(* IEC 61131-3 sources: Codesys/ddyut/src (part 2) *)

(* ---- FB_FountainSchedule.st ---- *)
(* ================================================================
   FB_FountainSchedule — Расписание Фонтана (свет + насосы)
   === ДДЮТ:ИЗМЕНЕНО (round 2) === У СВЕТА и НАСОСОВ теперь РАЗНОЕ
   число режимов и РАЗНАЯ кодировка — не путать порядок!

   СВЕТ (Light_Mode, UDINT, 4 положения):
     0 = АВТО   — включение по фиксированному расписанию
                  (Light_On_Hour/Minute_Weekday/Weekend), выключение
                  — общий Off_Hour/Minute (будни/выходные)
     1 = ВКЛ    — горит постоянно, не выключается никогда
     2 = ВЫКЛ   — не включается никогда
     3 = АСТРО  — включение по расчёту заката (Sunset_Hour/Minute
                  от FB_SunsetRelay), выключение — тот же общий
                  Off_Hour/Minute

   НАСОСЫ (Pump_Mode, UDINT, 3 положения — БЕЗ режима "Астро"):
     0 = АВТО   — включение по фиксированному расписанию
                  (Pump_On_Hour/Minute_Weekday/Weekend), выключение
                  — тот же общий Off_Hour/Minute
     1 = ВКЛ    — работает постоянно, не выключается никогда
     2 = ВЫКЛ   — не включается никогда

   === ДДЮТ:ИЗМЕНЕНО === Раньше (round 1) у обоих было по 4
   одинаковых положения (0=Астро,1=Авто,2=Вкл,3=Выкл), полная
   симметрия. По итогам практики решили, что насосам "Астро" не
   нужен — оставили только 3 положения, и заодно поменяли порядок
   у света (Авто теперь 0, Астро — последний, 3). Если переносишь
   в другой проект — ПЕРЕПРОВЕРЬ кодировку, она несимметричная.

   ВАЖНО: это ВНУТРЕННИЙ выбор — работает только когда ВНЕШНИЙ
   селектор узла (GVL_Fountain.iLightSelect / iPumpSelect, экран
   "Свет/Насосы") стоит в положении "Авто" (=2). При "Ручной пуск"
   (=0) и "Выкл" (=1) на внешнем селекторе — этот блок и его режимы
   вообще не участвуют в управлении DO1/DO9.

   ================================================================
   ФЛАГИ ВИДИМОСТИ ДЛЯ ЭКРАНА — единая схема имён:
   Объект_ЧтоПоказывает (Light_/Pump_ + ShowInputFields/
   ShowComputedTime/ShowAlwaysOnText/ShowAlwaysOffText)

   СВЕТ (4 положения, 0=Авто,1=Вкл,2=Выкл,3=Астро):
   Light_ShowInputFields  = TRUE при Режим=0 (Авто) — поля ручного
     ввода расписания (Light_On_Hour/Minute_Weekday/Weekend).
   Light_ShowComputedTime = TRUE при Режим=0 (Авто) ИЛИ Режим=3
     (Астро) — число результата (Light_On_Result_Hour/Minute).
   Light_ShowAlwaysOnText  = TRUE при Режим=1 (Вкл) — текст
     "Свет Вкл ручн".
   Light_ShowAlwaysOffText = TRUE при Режим=2 (Выкл) — текст
     "Свет Выкл ручн".

   НАСОСЫ (3 положения, 0=Авто,1=Вкл,2=Выкл — своя кодировка!):
   Pump_ShowInputFields  = TRUE при Режим=0 (Авто) — поля ручного
     ввода расписания (Pump_On_Hour/Minute_Weekday/Weekend).
   Pump_ShowComputedTime = TRUE при Режим=0 (Авто) — число
     результата. У насосов больше НЕТ режима "Астро" — этот флаг
     истинен только в одном положении, не в двух, как у света.
   Pump_ShowAlwaysOnText  = TRUE при Режим=1 (Вкл) — текст
     "Насосы Вкл ручн".
   Pump_ShowAlwaysOffText = TRUE при Режим=2 (Выкл) — текст
     "Насосы Выкл ручн".

   ---- ОБЩИЕ ПОЛЯ ВЫКЛЮЧЕНИЯ (Off_Result_Hour/Minute — результат,
   и Off_Hour/Minute_Weekday/Weekend — поля ручного ввода уставок) ----
   Актуальны (должны быть видны), если ХОТЯ БЫ ОДИН из двух объектов
   (свет ИЛИ насос) сейчас работает по времени — то есть находится
   в режиме, где Xxx_ShowComputedTime истинен. Если оба постоянно
   "Вкл"/"Выкл" — время выключения нигде не используется, поля
   можно скрыть.

   Off_Time_Visible = Light_ShowComputedTime ИЛИ Pump_ShowComputedTime

   Привязать «Видимость» ко ВСЕМ 6 полям сразу (один и тот же провод
   на несколько свойств «Видимость» — это нормально):
     Off_Result_Hour, Off_Result_Minute,
     Off_Hour_Weekday, Off_Minute_Weekday,
     Off_Hour_Weekend, Off_Minute_Weekend
   ================================================================ *)

FUNCTION_BLOCK FB_FountainSchedule

VAR_INPUT
    (* --- От FB_SunsetRelay --- *)
    Sunset_Auto         : BOOL;
    Sunset_Hour         : UDINT;
    Sunset_Minute       : UDINT;
    IsWeekend           : BOOL;

    (* --- Селектор режима СВЕТА: 0=Авто,1=Вкл,2=Выкл,3=Астро --- *)
    Light_Mode          : UDINT;

    (* --- Ручное расписание СВЕТА (режим 0=Авто): включение --- *)
    Light_On_Hour_Weekday   : UDINT;
    Light_On_Minute_Weekday : UDINT;
    Light_On_Hour_Weekend   : UDINT;
    Light_On_Minute_Weekend : UDINT;

    (* --- Выключение (общее для света и насосов) --- *)
    Off_Hour_Weekday    : UDINT;
    Off_Minute_Weekday  : UDINT;
    Off_Hour_Weekend    : UDINT;
    Off_Minute_Weekend  : UDINT;

    (* --- Селектор режима НАСОСОВ: 0=Авто,1=Вкл,2=Выкл (БЕЗ Астро) --- *)
    Pump_Mode                : UDINT;

    (* --- Ручное расписание НАСОСОВ (режим 0=Авто): включение --- *)
    Pump_On_Hour_Weekday    : UDINT;
    Pump_On_Minute_Weekday  : UDINT;
    Pump_On_Hour_Weekend    : UDINT;
    Pump_On_Minute_Weekend  : UDINT;

    (* --- Текущее время --- *)
    Sys_Hour            : UDINT;
    Sys_Minute          : UDINT;
END_VAR

VAR_OUTPUT
    Light_Out             : BOOL;   (* ВЫХОД на освещение (DO)                *)
    Pump_Out               : BOOL;   (* ВЫХОД на насосы фонтана (DO)           *)

    (* Итоговое время включения СВЕТА на сегодня — для экрана.
       В режимах 1/2 (Вкл/Выкл) содержит 0:00 (заглушка) — привязать
       видимость к Light_ShowComputedTime, чтобы не показывать её.  *)
    Light_On_Result_Hour   : UDINT;
    Light_On_Result_Minute : UDINT;

    (* Итоговое время включения НАСОСОВ на сегодня — для экрана.
       Аналогично, заглушка 0:00 в режимах 1/2 (Вкл/Выкл).          *)
    Pump_On_Result_Hour     : UDINT;
    Pump_On_Result_Minute   : UDINT;

    (* Единое время ВЫКЛЮЧЕНИЯ — общее поле для света и насосов *)
    Off_Result_Hour         : UDINT;
    Off_Result_Minute       : UDINT;

    (* --- Флаги видимости: СВЕТ (0=Авто,1=Вкл,2=Выкл,3=Астро) --- *)
    Light_ShowInputFields    : BOOL;  (* Режим=0(Авто) → поля ручного ввода *)
    Light_ShowComputedTime   : BOOL;  (* Режим=0(Авто) или 3(Астро) → число результата *)
    Light_ShowAlwaysOnText   : BOOL;  (* Режим=1(Вкл) → текст "Свет Вкл ручн" *)
    Light_ShowAlwaysOffText  : BOOL;  (* Режим=2(Выкл) → текст "Свет Выкл ручн" *)

    (* --- Флаги видимости: НАСОСЫ (0=Авто,1=Вкл,2=Выкл, своя кодировка) --- *)
    Pump_ShowInputFields     : BOOL;  (* Режим=0(Авто) → поля ручного ввода *)
    Pump_ShowComputedTime    : BOOL;  (* Режим=0(Авто) → число результата (Астро нет) *)
    Pump_ShowAlwaysOnText    : BOOL;  (* Режим=1(Вкл) → текст "Насосы Вкл ручн" *)
    Pump_ShowAlwaysOffText   : BOOL;  (* Режим=2(Выкл) → текст "Насосы Выкл ручн" *)

    (* Комбинированный флаг для полей времени ВЫКЛЮЧЕНИЯ фонтана
       (Off_Result_Hour/Minute И Off_Hour/Minute_Weekday/Weekend).
       TRUE если хотя бы один из объектов (свет ИЛИ насос) сейчас
       работает по времени.                                        *)
    Off_Time_Visible          : BOOL;
END_VAR

VAR
    now_total_min       : UDINT;
    light_on_min         : UDINT;
    light_off_min        : UDINT;
    pump_on_min           : UDINT;
    pump_off_min          : UDINT;
    off_today_min         : UDINT;  (* Общее время выключения на сегодня (мин) *)
END_VAR

(* ----------------------------------------------------------------
   Текущее время в минутах от 0:00
   ---------------------------------------------------------------- *)
now_total_min := Sys_Hour * 60 + Sys_Minute;

(* Общее время выключения на сегодня (будни/выходные) — используется
   и светом, и насосами, в любом режиме, где это осмысленно          *)
IF IsWeekend THEN
    off_today_min := Off_Hour_Weekend * 60 + Off_Minute_Weekend;
ELSE
    off_today_min := Off_Hour_Weekday * 60 + Off_Minute_Weekday;
END_IF;

(* ================================================================
   СВЕТ — 4 положения: 0=Авто,1=Вкл,2=Выкл,3=Астро
   ================================================================ *)

(* --- Light_Out по режиму --- *)
IF Light_Mode = 0 THEN
    (* АВТО: фиксированное расписание будни/выходные *)
    IF IsWeekend THEN
        light_on_min := Light_On_Hour_Weekend * 60 + Light_On_Minute_Weekend;
    ELSE
        light_on_min := Light_On_Hour_Weekday * 60 + Light_On_Minute_Weekday;
    END_IF;
    light_off_min := off_today_min;

    IF light_off_min > light_on_min THEN
        Light_Out := (now_total_min >= light_on_min) AND (now_total_min < light_off_min);
    ELSE
        Light_Out := (now_total_min >= light_on_min) OR (now_total_min < light_off_min);
    END_IF;

ELSIF Light_Mode = 1 THEN
    Light_Out := TRUE;   (* ВКЛ: горит постоянно *)

ELSIF Light_Mode = 3 THEN
    (* АСТРО: закат → общий Off *)
    light_on_min  := Sunset_Hour * 60 + Sunset_Minute;
    light_off_min := off_today_min;

    IF light_off_min > light_on_min THEN
        Light_Out := (now_total_min >= light_on_min) AND (now_total_min < light_off_min);
    ELSE
        Light_Out := (now_total_min >= light_on_min) OR (now_total_min < light_off_min);
    END_IF;

ELSE
    Light_Out := FALSE;  (* ВЫКЛ (2) или некорректное значение *)
END_IF;

(* --- Light_On_Result --- *)
IF Light_Mode = 0 THEN
    IF IsWeekend THEN
        Light_On_Result_Hour   := Light_On_Hour_Weekend;
        Light_On_Result_Minute := Light_On_Minute_Weekend;
    ELSE
        Light_On_Result_Hour   := Light_On_Hour_Weekday;
        Light_On_Result_Minute := Light_On_Minute_Weekday;
    END_IF;
ELSIF Light_Mode = 3 THEN
    Light_On_Result_Hour   := Sunset_Hour;
    Light_On_Result_Minute := Sunset_Minute;
ELSE
    Light_On_Result_Hour   := 0;   (* заглушка, режимы 1/2 (Вкл/Выкл) *)
    Light_On_Result_Minute := 0;
END_IF;

(* --- Флаги видимости СВЕТА --- *)
Light_ShowInputFields   := (Light_Mode = 0);
Light_ShowComputedTime  := (Light_Mode = 0) OR (Light_Mode = 3);
Light_ShowAlwaysOnText  := (Light_Mode = 1);
Light_ShowAlwaysOffText := (Light_Mode = 2);

(* ================================================================
   НАСОСЫ — 3 положения: 0=Авто,1=Вкл,2=Выкл (БЕЗ режима "Астро")
   ================================================================ *)

(* --- Pump_Out по режиму --- *)
IF Pump_Mode = 0 THEN
    (* АВТО: фиксированное расписание будни/выходные *)
    IF IsWeekend THEN
        pump_on_min := Pump_On_Hour_Weekend * 60 + Pump_On_Minute_Weekend;
    ELSE
        pump_on_min := Pump_On_Hour_Weekday * 60 + Pump_On_Minute_Weekday;
    END_IF;
    pump_off_min := off_today_min;

    IF pump_off_min > pump_on_min THEN
        Pump_Out := (now_total_min >= pump_on_min) AND (now_total_min < pump_off_min);
    ELSE
        Pump_Out := (now_total_min >= pump_on_min) OR (now_total_min < pump_off_min);
    END_IF;

ELSIF Pump_Mode = 1 THEN
    Pump_Out := TRUE;   (* ВКЛ: работает постоянно *)

ELSE
    Pump_Out := FALSE;  (* ВЫКЛ (2) или некорректное значение *)
END_IF;

(* --- Pump_On_Result --- *)
IF Pump_Mode = 0 THEN
    IF IsWeekend THEN
        Pump_On_Result_Hour   := Pump_On_Hour_Weekend;
        Pump_On_Result_Minute := Pump_On_Minute_Weekend;
    ELSE
        Pump_On_Result_Hour   := Pump_On_Hour_Weekday;
        Pump_On_Result_Minute := Pump_On_Minute_Weekday;
    END_IF;
ELSE
    Pump_On_Result_Hour   := 0;   (* заглушка, режимы 1/2 (Вкл/Выкл) *)
    Pump_On_Result_Minute := 0;
END_IF;

(* --- Флаги видимости НАСОСОВ --- *)
Pump_ShowInputFields   := (Pump_Mode = 0);
Pump_ShowComputedTime  := (Pump_Mode = 0);
Pump_ShowAlwaysOnText  := (Pump_Mode = 1);
Pump_ShowAlwaysOffText := (Pump_Mode = 2);

(* ================================================================
   ОБЩЕЕ ПОЛЕ Off_Result (время выключения, одно на экране)
   ================================================================ *)
Off_Result_Hour   := off_today_min / 60;
Off_Result_Minute := off_today_min MOD 60;

Off_Time_Visible := Light_ShowComputedTime OR Pump_ShowComputedTime;

(* ---- FB_Pump.st ---- *)
(* ============================================================ *)
(* FB_Pump — управление одним ПЧ ELHART (PUMP/MINI) по Modbus  *)
(* Проект ДДЮТ (на основе Fontan_V1 / Саки Пруд).               *)
(* === ДДЮТ:ИЗМЕНЕНО === Температура (блок 6) — без деления на  *)
(* 10 (регистр 0x0006 на ДДЮТ отдаёт целые °C). См. комментарий  *)
(* в блоке 6 ниже.                                               *)
(* ============================================================ *)

FUNCTION_BLOCK FB_Pump
VAR_INPUT
    eType      : E_PumpType;
    xDebugMode : BOOL;
    xCommError : BOOL;
    xCommUnstable : BOOL;

    xRunCmd      : BOOL;
    rFreqSetHz   : REAL;

    wStatus          : WORD;
    wFaultReg        : WORD;
    wFreqSetRead     : WORD;
    wFreqActual      : WORD;
    wCurrentActual   : WORD;
    wSpeedActual     : WORD;
    wDcVoltage       : WORD;
    wTemperature     : WORD;
    wVoltageActual   : WORD;
    wRuntimeHoursRaw : WORD;
    wAccTimeRawRead        : WORD;
    wDecTimeRawRead        : WORD;
    wMaxFreqRead           : WORD;
    wMinFreqRead           : WORD;
    wMotorRatedCurrentRead : WORD;
    wMotorRatedVoltageRead : WORD;
    wOverCurrentLevelRead  : WORD;
    wOverheatLevelRead     : WORD;
    wOverCurAccRead        : WORD;
    wOverCurrentTimeRead   : WORD;
    wOverVoltProtectRead   : WORD;

    rAccTime_Set            : REAL;
    rDecTime_Set            : REAL;
    rMaxFreq_Set            : REAL;
    rMinFreq_Set            : REAL;
    rMotorRatedCurrent_Set  : REAL;
    rMotorRatedVoltage_Set  : REAL;
    rOverCurrentLevel_A_Set : REAL;
    rOverCurrentTime_Set    : REAL;
    xOverVoltProtect_Set    : BOOL;
    iOverheatLevel_Set      : INT;
    iOverCurAcc_Set         : INT;
END_VAR
VAR_OUTPUT
    wCmd  : WORD;
    wFreq : WORD;
    wAccTimeRawWrite        : WORD;
    wDecTimeRawWrite        : WORD;
    wMaxFreqWrite           : WORD;
    wMinFreqWrite           : WORD;
    wMotorRatedCurrentWrite : WORD;
    wMotorRatedVoltageWrite : WORD;
    wOverCurrentLevelWrite  : WORD;
    wOverCurrentTimeWrite   : WORD;
    wOverVoltProtectWrite   : WORD;
    wOverheatLevelWrite     : WORD;
    wOverCurAccWrite        : WORD;

    xRun       : BOOL;
    xStop      : BOOL;
    xAlarm     : BOOL;
    sState     : WSTRING(50);
    sFaultText : WSTRING(100);
    sTypeText  : WSTRING(20);
    xReverse   : BOOL;

    rFreqSetActHz : REAL;
    rFreqActHz    : REAL;
    rCurrentActA  : REAL;
    rSpeedActRpm  : REAL;
    rDcVoltageV   : REAL;
    iTemperatureC : INT;
    rVoltageActV  : REAL;
    rRuntimeHours : REAL;
    rAccTime_Disp            : REAL;
    rDecTime_Disp            : REAL;
    rMaxFreq_Disp            : REAL;
    rMinFreq_Disp            : REAL;
    rMotorRatedCurrent_Disp  : REAL;
    rMotorRatedVoltage_Disp  : REAL;
    rOverCurrentLevel_A_Disp : REAL;
    iOverCurrentLevel_pct_Disp : INT;
    iOverheatLevel_Disp      : INT;
    iOverCurAcc_Disp         : INT;
    rOverCurrentTime_Disp    : REAL;
    xOverVoltProtect_Disp    : BOOL;
END_VAR
VAR
    rK_Freq         : REAL;
    rFreqLim        : REAL;
    xFaultActive    : BOOL;
    wCleanFaultCode : WORD;
    iFaultCode      : INT;
    rTmp : REAL;
    iTmp : INT;
END_VAR

(* ========================================================= *)
(* 1. Коэффициент пересчёта частоты                          *)
(* PUMP: 0,01 Гц → k=100 | MINI: 0,1 Гц → k=10               *)
(* ========================================================= *)
IF eType = E_PumpType.PUMP THEN
    rK_Freq   := 100.0;
    sTypeText := "EMD-PUMP";
ELSE
    rK_Freq   := 10.0;
    sTypeText := "EMD-MINI v2.1";
END_IF;

(* ========================================================= *)
(* 2. Команда управления и задание частоты (0x2000 / 0x2001) *)
(* ========================================================= *)
rFreqLim := rFreqSetHz;
IF rFreqLim < cMinFreq THEN rFreqLim := cMinFreq; END_IF;
IF rFreqLim > cMaxFreq THEN rFreqLim := cMaxFreq; END_IF;

IF xRunCmd THEN
    wCmd  := 16#000A;
    wFreq := REAL_TO_WORD(rFreqLim * rK_Freq);
ELSE
    wCmd  := 16#0009;
    wFreq := REAL_TO_WORD(rFreqLim * rK_Freq);
END_IF;

(* ========================================================= *)
(* 3. Нет связи → показать и выйти                           *)
(* ========================================================= *)
xStop := FALSE; xRun := FALSE; xAlarm := FALSE;
xReverse := FALSE; xFaultActive := FALSE;

IF xCommError OR xCommUnstable THEN
    xAlarm     := FALSE;
    xStop      := FALSE;
    xRun       := FALSE;
    sState     := "Нет связи с ПЧ";
    sFaultText := "Проверьте RS-485 / адрес / питание ПЧ";
    RETURN;
END_IF;

(* ========================================================= *)
(* 4. Состояние ПЧ по 0x001C                                *)
(* ========================================================= *)
CASE eType OF
    E_PumpType.PUMP:
        xReverse := (wStatus AND 16#0004) <> 0;
        IF (wStatus AND 16#0008) <> 0 THEN
            xAlarm := TRUE; xFaultActive := TRUE; sState := "Авария";
        ELSIF (wStatus AND 16#0001) <> 0 THEN
            xRun := TRUE;
            IF xReverse THEN sState := "Работа (реверс)"; ELSE sState := "Работа"; END_IF;
        ELSE
            xStop := TRUE; sState := "Стоп";
        END_IF;
    E_PumpType.MINI:
        xReverse := (wStatus AND 16#0001) <> 0;
        IF (wStatus AND 16#0002) <> 0 THEN
            xRun := TRUE;
            IF xReverse THEN sState := "Работа (реверс)"; ELSE sState := "Работа"; END_IF;
        ELSE
            xStop := TRUE; sState := "Стоп";
        END_IF;
END_CASE;

(* ========================================================= *)
(* 5. Разбор аварий                                         *)
(* ========================================================= *)
CASE eType OF
    E_PumpType.PUMP:
        IF (wFaultReg AND 16#8000) <> 0 THEN
            xAlarm := TRUE; xRun := FALSE; xStop := FALSE; sState := "Авария";
            wCleanFaultCode := wFaultReg AND 16#7FFF;
            sFaultText := F_FaultCodeToText(eType, wCleanFaultCode);
        ELSE
            sFaultText := "Нет ошибок";
        END_IF;
    E_PumpType.MINI:
        iFaultCode := WORD_TO_INT(wFaultReg);
        IF (iFaultCode > 63) AND ((iFaultCode < 88) OR (iFaultCode > 91)) THEN
            xAlarm := TRUE; xRun := FALSE; xStop := FALSE; sState := "Авария";
            sFaultText := F_FaultCodeToText(eType, wFaultReg);
        ELSE
            sFaultText := "Нет ошибок";
        END_IF;
END_CASE;

(* ========================================================= *)
(* 6. ЧТЕНИЕ реальных значений из ПЧ → _Disp (для показа)    *)
(* ========================================================= *)
rFreqSetActHz := WORD_TO_REAL(wFreqSetRead) / rK_Freq;
rFreqActHz    := WORD_TO_REAL(wFreqActual)  / rK_Freq;
rCurrentActA  := WORD_TO_REAL(wCurrentActual) / 10.0;
rSpeedActRpm  := WORD_TO_REAL(wSpeedActual);
rDcVoltageV   := WORD_TO_REAL(wDcVoltage) / 10.0;

(* === ДДЮТ:ИЗМЕНЕНО === Температура: БЕЗ деления на 10.       *)
(* На Саки регистр 0x0006 отдавал ×10 (0.1°C), на ДДЮТ — уже    *)
(* целые °C (та же марка ПЧ, но другая дискретность регистра —  *)
(* сверено на объекте: /10.0 давало 4°C вместо реальных 40°C).  *)
(* Если на твоём ПЧ регистр всё-таки ×10 — верни /10.0 обратно. *)
iTemperatureC := WORD_TO_INT(wTemperature);

rVoltageActV  := WORD_TO_REAL(wVoltageActual) / 10.0;
rRuntimeHours := WORD_TO_REAL(wRuntimeHoursRaw);

rAccTime_Disp           := WORD_TO_REAL(wAccTimeRawRead) / 10.0;
rDecTime_Disp           := WORD_TO_REAL(wDecTimeRawRead) / 10.0;
rMaxFreq_Disp           := WORD_TO_REAL(wMaxFreqRead) / rK_Freq;
rMinFreq_Disp           := WORD_TO_REAL(wMinFreqRead) / rK_Freq;
rMotorRatedCurrent_Disp := WORD_TO_REAL(wMotorRatedCurrentRead) / 10.0;
rMotorRatedVoltage_Disp := WORD_TO_REAL(wMotorRatedVoltageRead) / 10.0;
iOverCurrentLevel_pct_Disp := WORD_TO_INT(wOverCurrentLevelRead);
IF rMotorRatedCurrent_Disp > 0.0 THEN
    rOverCurrentLevel_A_Disp := (INT_TO_REAL(iOverCurrentLevel_pct_Disp) / 100.0)
                                 * rMotorRatedCurrent_Disp;
ELSE
    rOverCurrentLevel_A_Disp := 0.0;
END_IF;
iOverheatLevel_Disp := WORD_TO_INT(wOverheatLevelRead);
iOverCurAcc_Disp    := WORD_TO_INT(wOverCurAccRead);
rOverCurrentTime_Disp := WORD_TO_REAL(wOverCurrentTimeRead) / 10.0;
xOverVoltProtect_Disp := (wOverVoltProtectRead <> WORD#0);

(* ========================================================= *)
(* 7. ЗАДАНИЕ оператора → регистры ЗАПИСИ (_Set, с валидацией)*)
(* ========================================================= *)
rTmp := rAccTime_Set;
IF rTmp < cMinTime THEN rTmp := cMinTime; ELSIF rTmp > cMaxTime THEN rTmp := cMaxTime; END_IF;
wAccTimeRawWrite := REAL_TO_WORD(rTmp * 10.0);

rTmp := rDecTime_Set;
IF rTmp < cMinTime THEN rTmp := cMinTime; ELSIF rTmp > cMaxTime THEN rTmp := cMaxTime; END_IF;
wDecTimeRawWrite := REAL_TO_WORD(rTmp * 10.0);

rTmp := rMaxFreq_Set;
IF rTmp < 1.0 THEN rTmp := 1.0; ELSIF rTmp > cMaxFreq THEN rTmp := cMaxFreq; END_IF;
wMaxFreqWrite := REAL_TO_WORD(rTmp * rK_Freq);
rTmp := rMinFreq_Set;
IF rTmp < 0.0 THEN rTmp := 0.0; ELSIF rTmp > rMaxFreq_Set THEN rTmp := rMaxFreq_Set; END_IF;
wMinFreqWrite := REAL_TO_WORD(rTmp * rK_Freq);

rTmp := rMotorRatedVoltage_Set;
IF rTmp < 0.0 THEN rTmp := 0.0; ELSIF rTmp > cMaxVoltage THEN rTmp := cMaxVoltage; END_IF;
wMotorRatedVoltageWrite := REAL_TO_WORD(rTmp * 10.0);
rTmp := rMotorRatedCurrent_Set;
IF rTmp < 0.1 THEN rTmp := 0.1; ELSIF rTmp > cMaxCurrent THEN rTmp := cMaxCurrent; END_IF;
wMotorRatedCurrentWrite := REAL_TO_WORD(rTmp * 10.0);

IF rMotorRatedCurrent_Set > 0.0 THEN
    iTmp := REAL_TO_INT((rOverCurrentLevel_A_Set / rMotorRatedCurrent_Set) * 100.0);
ELSE
    iTmp := 0;
END_IF;
IF iTmp < 0 THEN iTmp := 0; ELSIF iTmp > 200 THEN iTmp := 200; END_IF;
wOverCurrentLevelWrite := INT_TO_WORD(iTmp);

rTmp := rOverCurrentTime_Set;
IF rTmp < 0.0 THEN rTmp := 0.0; END_IF;
CASE eType OF
    E_PumpType.PUMP: IF rTmp > 999.9 THEN rTmp := 999.9; END_IF;
    E_PumpType.MINI: IF rTmp > 5.0 THEN rTmp := 5.0; END_IF;
END_CASE;
wOverCurrentTimeWrite := REAL_TO_WORD(rTmp * 10.0);

IF xOverVoltProtect_Set THEN wOverVoltProtectWrite := 1; ELSE wOverVoltProtectWrite := 0; END_IF;

iTmp := iOverheatLevel_Set;
IF iTmp < cMinOverheat THEN iTmp := cMinOverheat; ELSIF iTmp > cMaxOverheat THEN iTmp := cMaxOverheat; END_IF;
wOverheatLevelWrite := INT_TO_WORD(iTmp);

iTmp := iOverCurAcc_Set;
IF iTmp < 0 THEN iTmp := 0; ELSIF iTmp > 200 THEN iTmp := 200; END_IF;
wOverCurAccWrite := INT_TO_WORD(iTmp);

(* ---- FB_SdSpaceGuard.st ---- *)
(* ============================================================ *)
(* FB_SdSpaceGuard — СТОРОЖ МЕСТА НА SD + УДАЛЕНИЕ САМОГО        *)
(*                   СТАРОГО МЕСЯЦА ЖУРНАЛОВ                     *)
(* ============================================================ *)
(* Ёмкость карты приходит на вход udiUsableMB: её определяет сам   *)
(* FB_SdCardSize (читает размер раздела у ядра), а если не вышло — *)
(* берётся номинал из выпадающего списка на экране (iSdCardSize).  *)
(*                                                               *)
(* ЧТО ДЕЛАЕТ ЗА ОДИН ЗАПУСК (фронт xTrigger):                    *)
(*   1. Обходит каталог журналов (DirOpen → DirList → DirClose):  *)
(*      считает, сколько занимают НАШИ журналы и сколько чужие,   *)
(*      и ищет САМЫЙ СТАРЫЙ месяц.                               *)
(*   2. Считает потолок:                                          *)
(*        квота = ёмкость карты − резерв 100 МБ − чужие файлы     *)
(*      То есть журналам достаётся ВСЯ карта, кроме резерва: на   *)
(*      32 ГБ это ~28,9 ГБ, на 2 ГБ ~1,7 ГБ. Ничего не пропадает. *)
(*   3. Если наши журналы переросли квоту — удаляет ТРИ файла     *)
(*      самого старого месяца и повторяет с пункта 1, пока не     *)
(*      уложится.                                                *)
(*                                                               *)
(* ⚠️ В квоту считается объём ТОЛЬКО наших файлов (прошедших       *)
(* разбор F_SdLogMonthKey), а чужие вычитаются из ёмкости — так    *)
(* чей-то архив на карте уменьшает наш потолок, но удалён быть не  *)
(* может. Содержимое ВЛОЖЕННЫХ папок не считается (DirList в       *)
(* глубину не ходит) — папку app.spk1xxm01 с загрузочным           *)
(* приложением (единицы МБ) перекрывает резерв в 100 МБ.           *)
(*                                                               *)
(* ЗАЩИТЫ ОТ УДАЛЕНИЯ ЛИШНЕГО:                                    *)
(*   • Удаляются только имена, ТОЧНО совпавшие с шаблоном         *)
(*     "<префикс>MM-YYYY.log" (разбор в F_SdLogMonthKey).         *)
(*   • Файл текущего месяца (в который идёт запись) не может быть *)
(*     удалён в принципе: кандидат обязан быть СТРОГО СТАРШЕ.     *)
(*   • Сравнение по числовому ключу YYYY*12+MM-1, а не по строке: *)
(*     12-2025 корректно старше 01-2026.                          *)
(*   • Каталоги (deDirEntry.xDirectory) пропускаются целиком.      *)
(*   • Если обход каталога оборвался по лимиту — «самый старый»   *)
(*     недостоверен, и не удаляется НИЧЕГО.                       *)
(*                                                               *)
(* ЕСЛИ УДАЛЯТЬ УЖЕ НЕЧЕГО, А КВОТА ВСЁ РАВНО ПРЕВЫШЕНА           *)
(* (вся история — это один текущий месяц, раздутый дребезгом      *)
(* аварий), поднимается xQuotaStop, и PRG_AlarmLogSD ПРЕКРАЩАЕТ   *)
(* запись на карту. Это последний рубеж: карта не переполнится    *)
(* никогда, фонтан работает, журналы на экране ведутся как        *)
(* обычно. Снимается само при смене месяца, когда раздутый файл   *)
(* станет прошлым и его можно будет удалить. Человек не нужен.    *)
(*                                                               *)
(* ЕДИНИЦЫ. Внутри всё в КиБ (1024 байта), наружу и в пороги — в   *)
(* МиБ (1024 КиБ = 1 048 576 байт). 100 МБ = 104 857 600 байт.    *)
(* Деление целочисленное: оценка свободного всегда чуть ЗАНИЖЕНА, *)
(* то есть чистка срабатывает на доли мегабайта РАНЬШЕ.           *)
(*                                                               *)
(* ФБ асинхронный: один запуск растянут на много циклов ПЛК       *)
(* (каждый ФБ CAA File требует минимум цикл). Пока xBusy = TRUE,  *)
(* PRG_AlarmLogSD не начинает новую запись строки.                *)
(* ============================================================ *)
FUNCTION_BLOCK FB_SdSpaceGuard
VAR_INPUT
    xTrigger      : BOOL;        (* ФРОНТ — выполнить проверку *)
    xForce        : BOOL;        (* уровень, читается при старте: удалить    *)
                                 (* самый старый месяц БЕЗ проверок. Ставится*)
                                 (* автоматически, когда запись на карту не  *)
                                 (* проходит подряд несколько раз (значит,   *)
                                 (* карта реально полна — например, номинал  *)
                                 (* в списке выбран больше настоящего).      *)
    sDir          : STRING(80);  (* каталог журналов, БЕЗ '/' в конце *)
    sPrefix1      : STRING(20);  (* 'alarms-' *)
    sPrefix2      : STRING(20);  (* 'pump_changes-' *)
    sPrefix3      : STRING(20);  (* 'setpoints-' *)
    udiUsableMB   : UDINT;       (* полезная ёмкость карты, МиБ *)
    udiFreeMinMB  : UDINT;       (* резерв свободного места, МиБ (100) *)
    iCurYear      : INT;         (* текущий год  журнала (2000..2199) *)
    iCurMonth     : INT;         (* текущий месяц журнала (1..12) *)
END_VAR
VAR_OUTPUT
    xBusy            : BOOL;
    xDone            : BOOL;      (* импульс 1 цикл по завершении запуска *)
    xQuotaStop       : BOOL;      (* ⛔ писать на SD больше нельзя *)
    udiQuotaMB       : UDINT;     (* сколько реально отдано журналам, МиБ *)
    udiOursMB        : UDINT;     (* занято НАШИМИ журналами, МиБ *)
    udiUsedMB        : UDINT;     (* занято всеми файлами каталога, МиБ *)
    udiForeignMB     : UDINT;     (* занято чужими файлами рядом, МиБ *)
    udiOldestMB      : UDINT;     (* объём самого старого месяца, МиБ *)
    xNothingToDelete : BOOL;      (* чистить надо, а удалять нечего *)
    xFault           : BOOL;      (* карта/каталог недоступны, скан сорван *)
    iDeletedTotal    : INT;       (* удалено файлов с момента старта ПЛК *)
    iDeletedLast     : INT;       (* удалено за последний запуск *)
    sLastDeleted     : STRING(80);(* что удалили последним *)
    iFilesSeen       : INT;       (* файлов в каталоге на последнем скане *)
END_VAR
VAR CONSTANT
    cMaxRounds  : INT := 24;      (* не больше 24 месяцев за один запуск *)
    cMaxEntries : INT := 500;     (* страховка от бесконечного DirList *)
END_VAR
VAR
    iSt        : INT;
    xTrigPrev  : BOOL;
    iRound     : INT;

    fbDirOpen  : FILE.DirOpen;
    fbDirList  : FILE.DirList;
    fbDirClose : FILE.DirClose;
    fbDelete   : FILE.Delete;
    hDir       : FILE.CAA.HANDLE;

    udiUsedKB    : UDINT;   (* все файлы каталога, КиБ (диагностика) *)
    udiOursKB    : UDINT;   (* только наши журналы, КиБ (для квоты) *)
    udiEntryKB   : UDINT;
    udiCurKey    : UDINT;
    udiOldKey    : UDINT;
    udiOldestKB  : UDINT;   (* объём файлов самого старого месяца, КиБ *)
    udiKey       : UDINT;
    xFoundOld    : BOOL;
    xForceRun    : BOOL;
    xOverQuota   : BOOL;
    iEntries     : INT;
    sEntry       : STRING(255);

    iOldYear        : INT;
    iOldMonth       : INT;
    iDelIdx         : INT;
    iDelOkThisRound : INT;
    sDelPath        : STRING(80);
END_VAR

(* ============================================================ *)
(* ЗАПУСК ПО ФРОНТУ                                             *)
(* ============================================================ *)
IF xTrigger AND NOT xTrigPrev AND iSt = 0 THEN
    xForceRun := xForce;      (* режим запуска фиксируем в момент старта *)
    iSt := 10;
END_IF;
xTrigPrev := xTrigger;

xDone := FALSE;
xBusy := (iSt <> 0);

CASE iSt OF

    0:  (* IDLE *)
        ;

    10: (* НАЧАЛО ЗАПУСКА *)
        iRound           := 0;
        iDeletedLast     := 0;
        xNothingToDelete := FALSE;
        xFault           := FALSE;
        iSt := 11;

    11: (* НАЧАЛО РАУНДА — подготовка скана каталога *)
        IF iCurYear < 2000 OR iCurYear > 2199 OR iCurMonth < 1 OR iCurMonth > 12 THEN
            (* без достоверного «сегодня» нельзя понять, какой месяц    *)
            (* трогать нельзя → не удаляем НИЧЕГО                        *)
            xFault := TRUE;
            iSt := 90;
        ELSE
            udiCurKey    := INT_TO_UDINT(iCurYear) * 12 + INT_TO_UDINT(iCurMonth) - 1;
            udiUsedKB    := 0;
            udiOursKB    := 0;
            udiOldKey    := 0;
            udiOldestKB  := 0;
            xFoundOld    := FALSE;
            iEntries     := 0;
            iSt := 12;
        END_IF;

    12: (* DirOpen *)
        fbDirOpen(xExecute := TRUE, sDirName := sDir);
        IF fbDirOpen.xDone THEN
            hDir := fbDirOpen.hDir;
            fbDirOpen(xExecute := FALSE);
            iSt := 13;
        ELSIF fbDirOpen.xError THEN
            fbDirOpen(xExecute := FALSE);
            xFault := TRUE;          (* карты нет / каталог недоступен *)
            iSt := 90;
        END_IF;

    13: (* DirList — по ОДНОЙ записи за вызов, до NO_MORE_ENTRIES *)
        fbDirList(xExecute := TRUE, hDir := hDir);
        IF fbDirList.xDone THEN
            IF NOT fbDirList.deDirEntry.xDirectory THEN
                sEntry := fbDirList.deDirEntry.sEntry;

                (* объём: округляем вверх до КиБ — оценка занятого места     *)
                (* получается чуть больше реальной суммы байт, это в нужную  *)
                (* сторону (реальный расход по кластерам FAT ещё больше)     *)
                udiEntryKB := (fbDirList.deDirEntry.szSize / 1024) + 1;
                udiUsedKB  := udiUsedKB + udiEntryKB;

                (* наш ли это файл и за какой месяц *)
                udiKey := F_SdLogMonthKey(sEntry, sPrefix1);
                IF udiKey = 0 THEN udiKey := F_SdLogMonthKey(sEntry, sPrefix2); END_IF;
                IF udiKey = 0 THEN udiKey := F_SdLogMonthKey(sEntry, sPrefix3); END_IF;

                IF udiKey > 0 THEN
                    (* КВОТА считается только по НАШИМ файлам *)
                    udiOursKB := udiOursKB + udiEntryKB;

                    (* кандидат на удаление — только СТРОГО СТАРШЕ текущего *)
                    IF udiKey < udiCurKey THEN
                        IF NOT xFoundOld OR udiKey < udiOldKey THEN
                            (* нашли месяц старее — объём считаем заново *)
                            udiOldKey   := udiKey;
                            udiOldestKB := udiEntryKB;
                            xFoundOld   := TRUE;
                        ELSIF udiKey = udiOldKey THEN
                            (* ещё один файл того же самого старого месяца *)
                            udiOldestKB := udiOldestKB + udiEntryKB;
                        END_IF;
                    END_IF;
                END_IF;
            END_IF;

            iEntries := iEntries + 1;
            fbDirList(xExecute := FALSE);
            IF iEntries >= cMaxEntries THEN
                (* Каталог не дочитан до конца → «самый старый месяц»         *)
                (* определён по неполному списку и может быть НЕ самым старым. *)
                (* Удалять по недостоверным данным нельзя: закрываем каталог   *)
                (* и выходим с аварией. 500 файлов — это ~13 лет журналов,     *)
                (* столько бывает только если на карте лежит что-то чужое.     *)
                xFault := TRUE;
                iSt := 14;
            END_IF;
        ELSIF fbDirList.xError THEN
            (* штатное окончание обхода = ERROR.NO_MORE_ENTRIES *)
            fbDirList(xExecute := FALSE);
            iSt := 14;
        END_IF;

    14: (* DirClose — закрыть каталог НАДО в любом случае, даже по аварии *)
        fbDirClose(xExecute := TRUE, hDir := hDir);
        IF fbDirClose.xDone OR fbDirClose.xError THEN
            fbDirClose(xExecute := FALSE);
            iFilesSeen := iEntries;
            IF xFault THEN
                iSt := 90;      (* скан недостоверен — ничего не удаляем *)
            ELSE
                iSt := 20;
            END_IF;
        END_IF;

    20: (* ОЦЕНКА: КВОТА *)
        udiUsedMB   := udiUsedKB / 1024;
        udiOursMB   := udiOursKB / 1024;
        udiOldestMB := udiOldestKB / 1024;

        (* --- сколько можно отдать журналам ---                          *)
        (* Вся карта минус резерв минус ЧУЖИЕ файлы, лежащие рядом в том  *)
        (* же каталоге (например, распакованное загрузочное приложение).  *)
        (* ⚠️ Содержимое ВЛОЖЕННЫХ папок не считается — DirList в глубину  *)
        (* не ходит. Папку app.spk1xxm01 с проектом (единицы МБ) с лихвой  *)
        (* перекрывает резерв в 100 МБ.                                   *)
        udiForeignMB := udiUsedMB - udiOursMB;
        IF udiUsableMB > (udiFreeMinMB + udiForeignMB) THEN
            udiQuotaMB := udiUsableMB - udiFreeMinMB - udiForeignMB;
        ELSE
            udiQuotaMB := 0;    (* чужие файлы съели всё — чистимся до дна *)
        END_IF;

        (* --- превышен ли потолок --- *)
        xOverQuota := (udiOursMB > udiQuotaMB);

        iSt := 30;

    30: (* РЕШЕНИЕ: чистить или нет *)
        IF xForceRun OR xOverQuota THEN
            IF xFoundOld THEN
                iOldYear        := UDINT_TO_INT(udiOldKey / 12);
                iOldMonth       := UDINT_TO_INT(udiOldKey MOD 12) + 1;
                iDelIdx         := 1;
                iDelOkThisRound := 0;
                iSt := 40;
            ELSE
                (* Старше текущего месяца ничего нет. Если при этом превышена *)
                (* наша собственная квота — единственный оставшийся способ не *)
                (* переполнить карту — перестать писать. Снимется само на     *)
                (* следующем месяце.                                          *)
                xNothingToDelete := TRUE;
                xQuotaStop       := xOverQuota;
                iSt := 90;
            END_IF;
        ELSE
            (* всё в норме — снимаем запрет записи, если он был *)
            xNothingToDelete := FALSE;
            xQuotaStop       := FALSE;
            iSt := 90;
        END_IF;

    40: (* ИМЯ ОЧЕРЕДНОГО ФАЙЛА САМОГО СТАРОГО МЕСЯЦА *)
        CASE iDelIdx OF
            1: sDelPath := F_SdLogPath(sDir, sPrefix1, iOldYear, iOldMonth);
            2: sDelPath := F_SdLogPath(sDir, sPrefix2, iOldYear, iOldMonth);
            3: sDelPath := F_SdLogPath(sDir, sPrefix3, iOldYear, iOldMonth);
        END_CASE;
        iSt := 41;

    41: (* УДАЛЕНИЕ *)
        fbDelete(xExecute := TRUE, sFileName := sDelPath);
        IF fbDelete.xDone THEN
            fbDelete(xExecute := FALSE);
            iDeletedLast    := iDeletedLast + 1;
            iDeletedTotal   := iDeletedTotal + 1;
            iDelOkThisRound := iDelOkThisRound + 1;
            sLastDeleted    := sDelPath;
            iSt := 42;
        ELSIF fbDelete.xError THEN
            (* файла за этот месяц могло не быть (например, уставки никто    *)
            (* не менял) — это норма, просто идём дальше                     *)
            fbDelete(xExecute := FALSE);
            iSt := 42;
        END_IF;

    42: (* СЛЕДУЮЩИЙ ФАЙЛ ИЛИ СЛЕДУЮЩИЙ РАУНД *)
        IF iDelIdx < 3 THEN
            iDelIdx := iDelIdx + 1;
            iSt := 40;
        ELSE
            iRound    := iRound + 1;
            xForceRun := FALSE;      (* аварийный форс = ровно один месяц *)
            IF iDelOkThisRound = 0 THEN
                (* Скан этот месяц нашёл, а удалить не вышло НИ ОДНОГО файла: *)
                (* карта только для чтения / вынута / имя на ФС отличается     *)
                (* регистром. Повторять раунды бессмысленно — они будут снова  *)
                (* находить тот же месяц. Выходим с аварией, чтобы это увидели.*)
                xFault := TRUE;
                iSt := 90;
            ELSIF iRound >= cMaxRounds THEN
                iSt := 90;
            ELSE
                iSt := 11;           (* пересчитать и, если надо, ещё раз *)
            END_IF;
        END_IF;

    90: (* КОНЕЦ ЗАПУСКА *)
        xDone := TRUE;
        iSt   := 0;

END_CASE;

(* ---- FB_SunsetRelay.st ---- *)
(* ============================================================
   FB_SunsetRelay — Астрономическое реле (расчёт заката)
   === ДДЮТ:ПОРТИРОВАНО (v2, точность до 1 мин) ===
   Единственное техническое отличие от твоего исходника (OwenLogic):
     SYS.COS/SYS.SIN/SYS.TAN/SYS.ACOS → COS/SIN/TAN/ACOS
     (в CODESYS это стандартные функции IEC 61131-3 без префикса
     SYS. — префикс есть только в библиотеке OwenLogic).
   Вся математика, включая поправку на рефракцию (90.833°) и
   алгоритм Зеллера — БЕЗ ИЗМЕНЕНИЙ, как в твоём исходнике.
   Логика:
   - Расчёт времени заката по долготе/широте/часовому поясу
   - Ручная коррекция ±минут (местность: море/горы/рельеф)
   - Выход «Sunset_Auto» = TRUE от заката до времени отключения
   - Точность расчёта: ±1-3 минуты (алгоритм NOAA/Spencer с поправкой
     на атмосферную рефракцию и радиус диска Солнца, угол зенита
     90.833°). Сверено с независимыми источниками для трёх городов
     на 12 месяцев вперёд.
   - Определение будни/выходной (алгоритм Зеллера) — для выбора
     своей пары Off_Hour/Off_Minute, а также выдаётся наружу
     (IsWeekend) для использования в FB_FountainSchedule, чтобы
     не дублировать расчёт дня недели в другом блоке.
   - Доп. выход: сколько осталось до следующей смены состояния

   ВАЖНО: Sunset_Auto — это ТОЛЬКО автоматический расчёт по закату.
   Финальное управление светом (авто/ручной режим) находится в
   отдельном блоке FB_FountainSchedule — туда подаётся Sunset_Auto
   как один из входов.
   ============================================================ *)

FUNCTION_BLOCK FB_SunsetRelay

VAR_INPUT
    (* --- Геокоординаты с экрана --- *)
    Latitude        : REAL;   (* Широта, градусы (пример: 44.59 = Севастополь)  *)
    Longitude       : REAL;   (* Долгота, градусы (пример: 33.52 = Севастополь) *)
    TimeZone        : REAL;   (* Часовой пояс, знаковый! ← выход FB_TimeZoneSelect *)

    (* --- Коррекция заката --- *)
    Sunset_Correct  : UDINT;  (* Ручная коррекция заката, минут (0..60)  *)
    Sunset_Earlier   : BOOL;  (* Направление: TRUE = раньше, FALSE = позже *)

    (* --- Настройки отключения: раздельно будни/выходные --- *)
    Off_Hour_Weekday   : UDINT;  (* Час отключения, будний день      *)
    Off_Minute_Weekday : UDINT;  (* Минута отключения, будний день   *)
    Off_Hour_Weekend   : UDINT;  (* Час отключения, выходной день    *)
    Off_Minute_Weekend : UDINT;  (* Минута отключения, выходной день *)

    (* --- Системное время (привязка к RTC ПР200) --- *)
    Sys_Year        : UDINT;  (* Год (2026)                              *)
    Sys_Month       : UDINT;  (* Месяц (1..12)                           *)
    Sys_Day         : UDINT;  (* День (1..31)                            *)
    Sys_Hour        : UDINT;  (* Часы (0..23)                            *)
    Sys_Minute      : UDINT;  (* Минуты (0..59)                          *)
    Sys_Sec         : UDINT;  (* Секунды (0..59) — для точности          *)
END_VAR

VAR_OUTPUT
    Sunset_Auto     : BOOL;   (* Автоматический расчёт: 1 = должно гореть *)
    Sunset_Hour     : UDINT;  (* Рассчитанный час заката (для экрана)    *)
    Sunset_Minute   : UDINT;  (* Рассчитанная минута заката (для экрана) *)
    DayOfYear       : UDINT;  (* Порядковый день года (диагностика)      *)
    Err_Coord       : BOOL;   (* Ошибка координат (широта за пределами)  *)
    IsWeekend       : BOOL;   (* TRUE = суббота/воскресенье. Выдаётся
                                  наружу для FB_FountainSchedule           *)

    (* --- Сколько осталось до следующего включения --- *)
    Time_Left_H     : UDINT;  (* Осталось ждать: часы                    *)
    Time_Left_M     : UDINT;  (* Осталось ждать: минуты (0–59)           *)
END_VAR

VAR
    (* --- Внутренние переменные расчёта заката --- *)
    i               : UDINT;
    doy             : UDINT;
    lat_rad         : REAL;
    gamma           : REAL;
    eqtime          : REAL;
    decl            : REAL;
    ha              : REAL;
    sunset_utc      : REAL;
    sunset_local    : REAL;
    sunset_total_min : UDINT;
    off_total_min   : UDINT;
    now_total_min   : UDINT;
    diff_min        : UDINT;
    pi              : REAL;
    two_pi          : REAL;
    deg_to_rad      : REAL;
    rad_to_deg      : REAL;
    temp_real       : REAL;
    sunset_corr_real : REAL;
    days_in_month   : ARRAY[1..12] OF UDINT;

    (* --- Внутренние переменные расчёта дня недели (алгоритм Зеллера) --- *)
    zm              : UDINT;  (* Месяц с коррекцией (янв/фев → 13/14 пред. года) *)
    zy              : UDINT;  (* Год с коррекцией                         *)
    zK              : UDINT;  (* Год внутри века (00-99)                  *)
    zJ              : UDINT;  (* Век (число столетий)                     *)
    zh              : UDINT;  (* Результат: 0=Сб,1=Вс,2=Пн,3=Вт,4=Ср,5=Чт,6=Пт *)
END_VAR

(* ============================================================
   ОПРЕДЕЛЕНИЕ ДНЯ НЕДЕЛИ (алгоритм Зеллера, григорианский календарь)
   Выполняется ВСЕГДА, независимо от Err_Coord — не зависит от
   координат, нужно для выбора Off_Hour/Off_Minute и для выдачи
   IsWeekend наружу.
   ============================================================ *)
IF Sys_Month < 3 THEN
    zm := Sys_Month + 12;
    zy := Sys_Year - 1;
ELSE
    zm := Sys_Month;
    zy := Sys_Year;
END_IF;

zK := zy MOD 100;
zJ := zy / 100;

zh := (Sys_Day + (13 * (zm + 1)) / 5 + zK + zK / 4 + zJ / 4 + 5 * zJ) MOD 7;

IsWeekend := (zh = 0) OR (zh = 1);   (* 0=суббота, 1=воскресенье *)

(* Выбор пары Off_Hour/Off_Minute по дню недели *)
IF IsWeekend THEN
    off_total_min := Off_Hour_Weekend * 60 + Off_Minute_Weekend;
ELSE
    off_total_min := Off_Hour_Weekday * 60 + Off_Minute_Weekday;
END_IF;

(* ============================================================
   ТЕЛО БЛОКА — РАСЧЁТ ЗАКАТА (АЛГОРИТМ NOAA)
   ============================================================ *)

pi := 3.14159265;
two_pi := 6.2831853;
deg_to_rad := pi / 180.0;
rad_to_deg := 180.0 / pi;

days_in_month[1] := 31;
days_in_month[2] := 28;
days_in_month[3] := 31;
days_in_month[4] := 30;
days_in_month[5] := 31;
days_in_month[6] := 30;
days_in_month[7] := 31;
days_in_month[8] := 31;
days_in_month[9] := 30;
days_in_month[10] := 31;
days_in_month[11] := 30;
days_in_month[12] := 31;

(* --- 1. Проверка координат --- *)
Err_Coord := (Latitude < -90.0) OR (Latitude > 90.0)
          OR (Longitude < -180.0) OR (Longitude > 180.0);

IF Err_Coord THEN
    Sunset_Auto := FALSE;
    Sunset_Hour := 0;
    Sunset_Minute := 0;
    DayOfYear := 0;
    Time_Left_H := 0;
    Time_Left_M := 0;

ELSE
    (* --- 2. День года --- *)
    doy := 0;
    FOR i := 1 TO 12 DO
        IF i < Sys_Month THEN
            doy := doy + days_in_month[i];
        END_IF;
    END_FOR;
    doy := doy + Sys_Day;

    IF (Sys_Year MOD 4 = 0) THEN
        IF (Sys_Year MOD 100 <> 0) OR (Sys_Year MOD 400 = 0) THEN
            IF Sys_Month > 2 THEN
                doy := doy + 1;
            END_IF;
        END_IF;
    END_IF;
    DayOfYear := doy;

    (* --- 3. Годовой угол (гамма) --- *)
    gamma := two_pi * UDINT_TO_REAL(doy - 1) / 365.0;

    (* --- 4. Уравнение времени (eqtime), минуты --- *)
    eqtime := 229.18 * (0.000075
             + 0.001868 * COS(gamma)
             - 0.032077 * SIN(gamma)
             - 0.014615 * COS(2.0 * gamma)
             - 0.040849 * SIN(2.0 * gamma));

    (* --- 5. Склонение Солнца (decl), радианы --- *)
    decl := 0.006918
          - 0.399912 * COS(gamma)
          + 0.070257 * SIN(gamma)
          - 0.006758 * COS(2.0 * gamma)
          + 0.000907 * SIN(2.0 * gamma)
          - 0.002697 * COS(3.0 * gamma)
          + 0.00148  * SIN(3.0 * gamma);

    (* --- 6. Часовой угол заката (ha), радианы ---
       Угол зенита 90.833° (не 90°!) — стандартная поправка на
       атмосферную рефракцию (~34') + видимый радиус диска Солнца
       (~16'). Без неё расчёт даёт закат на 3-7 мин раньше реального
       (сверено с независимыми таблицами для Севастополя, Краснодара,
       Москвы на 12 месяцев вперёд — после поправки разброс ±1-3 мин).
       ---------------------------------------------------------------- *)
    lat_rad := Latitude * deg_to_rad;
    temp_real := COS(90.833 * deg_to_rad) / (COS(lat_rad) * COS(decl))
                 - TAN(lat_rad) * TAN(decl);

    IF temp_real > 1.0 THEN
        ha := 0.0;
    ELSIF temp_real < -1.0 THEN
        ha := pi;
    ELSE
        ha := ACOS(temp_real);
    END_IF;

    (* --- 7. Закат в UTC, часы --- *)
    sunset_utc := 12.0 + (ha * rad_to_deg / 15.0) - (eqtime / 60.0) - (Longitude / 15.0);

    (* --- 8. Перевод в местное время --- *)
    sunset_local := sunset_utc + TimeZone;  (* TimeZone уже REAL, конверсия не нужна *)
    IF sunset_local < 0.0 THEN
        sunset_local := sunset_local + 24.0;
    END_IF;
    IF sunset_local >= 24.0 THEN
        sunset_local := sunset_local - 24.0;
    END_IF;

    (* --- 9. Применение ручной коррекции --- *)
    sunset_corr_real := UDINT_TO_REAL(Sunset_Correct) / 60.0;
    IF Sunset_Earlier THEN
        sunset_local := sunset_local - sunset_corr_real;
    ELSE
        sunset_local := sunset_local + sunset_corr_real;
    END_IF;

    IF sunset_local < 0.0 THEN
        sunset_local := sunset_local + 24.0;
    END_IF;
    IF sunset_local >= 24.0 THEN
        sunset_local := sunset_local - 24.0;
    END_IF;

    (* --- 10. Результат в часы/минуты — ПЕРЕПИСАНО (найден баг) --- *)
    (* БЫЛО: Sunset_Hour считался ОТДЕЛЬНО через REAL_TO_UDINT(sunset_local),*)
    (* а минуты — как остаток (sunset_local - Sunset_Hour) * 60. Проблема: *)
    (* REAL_TO_UDINT в CODESYS ОКРУГЛЯЕТ, а не отбрасывает дробную часть.  *)
    (* Если дробная часть часа была, например, 0.5527 — округление даёт    *)
    (* ЧАС НА ЕДИНИЦУ БОЛЬШЕ, а остаток для минут уходит В ОТРИЦАТЕЛЬНОЕ   *)
    (* число — которое тут же ломается при попытке положить его в UDINT   *)
    (* (беззнаковый тип), давая переполнение на ~4 миллиарда. Дальше это   *)
    (* переполнение триггерит "IF >= 60" и добавляет ЕЩЁ +1 к часу — так   *)
    (* 20:33 превращалось в 22 часа, а -87 минут "просвечивали" через      *)
    (* UDINT_TO_INT при отображении на экране (типичный пример: 20.5527ч  *)
    (* → час округлился до 21, остаток -26.84 мин → переполнение →        *)
    (* +1 к часу = 22, младшие 16 бит переполненного числа = -87).        *)
    (*                                                                    *)
    (* СТАЛО: переводим время заката сразу в ЦЕЛЫЕ МИНУТЫ ОДНИМ действием  *)
    (* (без разделения на час+остаток), потом делим нацело — так          *)
    (* отрицательное промежуточное значение в принципе невозможно.        *)
    sunset_total_min := REAL_TO_UDINT(sunset_local * 60.0);
    (* На случай если округление дало ровно 1440 (24:00 = начало следующих*)
    (* суток) — переносим на 0:00.                                        *)
    IF sunset_total_min >= 1440 THEN
        sunset_total_min := sunset_total_min - 1440;
    END_IF;
    Sunset_Hour   := sunset_total_min / 60;
    Sunset_Minute := sunset_total_min MOD 60;

    (* --- 11. Время заката в минутах от 0:00 (уже посчитано выше) --- *)

    (* --- 12. Текущее время в минутах от 0:00 --- *)
    now_total_min := Sys_Hour * 60 + Sys_Minute;

    (* off_total_min уже выбран выше (будни/выходной) *)

    (* --- 14. ЛОГИКА ВКЛЮЧЕНИЯ/ОТКЛЮЧЕНИЯ --- *)
    IF off_total_min > sunset_total_min THEN
        Sunset_Auto := (now_total_min >= sunset_total_min) AND (now_total_min < off_total_min);
    ELSE
        Sunset_Auto := (now_total_min >= sunset_total_min) OR (now_total_min < off_total_min);
    END_IF;

    (* --- 15. ВРЕМЯ ДО СЛЕДУЮЩЕГО ЗАКАТА --- *)
    IF now_total_min < sunset_total_min THEN
        diff_min := sunset_total_min - now_total_min;
    ELSE
        diff_min := (1440 - now_total_min) + sunset_total_min;
    END_IF;

    Time_Left_H := diff_min / 60;
    Time_Left_M := diff_min MOD 60;

END_IF;

(* ---- FB_TimeZoneSelect.st ---- *)
(* ================================================================
   FB_TimeZoneSelect — Выбор часового пояса комбобоксом
   === ДДЮТ:НОВЫЙ ФАЙЛ === Без технических изменений — синтаксис
   уже совместим с CODESYS 3.5 (нет SYS.* функций OwenLogic).

   ChoseTimeZone — индекс 0-23 с экрана (Текстовый список).
   Линейная зависимость: TimeZone = ChoseTimeZone - 11.
   ChoseTimeZone = 14 → TimeZone = +3 (Москва) — ЗНАЧЕНИЕ ПО
   УМОЛЧАНИЮ. Если оператор ничего не выберет — расчёт всё равно
   будет верным для объекта в РФ/Крыму, а не съедет на Гринвич.

   На экране создать «Текстовый список», привязанный к
   ChoseTimeZone, со строками:
   0  → "-11 Паго-Паго"
   1  → "-10 Гонолулу"
   2  → "-9  Анкоридж"
   3  → "-8  Лос-Анджелес"
   4  → "-7  Денвер"
   5  → "-6  Мехико"
   6  → "-5  Нью-Йорк"
   7  → "-4  Сантьяго"
   8  → "-3  Буэнос-Айрес"
   9  → "-2  Норонья"
   10 → "-1  Азорские о-ва"
   11 → "0   Лондон"
   12 → "+1  Берлин"
   13 → "+2  Калининград"
   14 → "+3  Москва"           ← ЗНАЧЕНИЕ ПО УМОЛЧАНИЮ
   15 → "+4  Самара"
   16 → "+5  Екатеринбург"
   17 → "+6  Омск"
   18 → "+7  Красноярск"
   19 → "+8  Иркутск"
   20 → "+9  Якутск"
   21 → "+10 Владивосток"
   22 → "+11 Магадан"
   23 → "+12 Камчатка"
   ================================================================ *)

FUNCTION_BLOCK FB_TimeZoneSelect
VAR_INPUT
    ChoseTimeZone   : UDINT;  (* Индекс выбора, 0-23. По умолчанию 14=Москва *)
END_VAR
VAR_OUTPUT
    TimeZone        : REAL;   (* → вход TimeZone в FB_SunsetRelay             *)
END_VAR
VAR
    idx             : UDINT;  (* Рабочая копия для проверки диапазона        *)
END_VAR

(* Защита от некорректного значения (>23) — откат на Москву (14) *)
IF ChoseTimeZone > 23 THEN
    idx := 14;
ELSE
    idx := ChoseTimeZone;
END_IF;

(* Линейное преобразование: индекс 0..23 → смещение -11..+12 *)
TimeZone := UDINT_TO_REAL(idx) - 11.0;

END_FUNCTION_BLOCK

(* ---- PLC_PRG.st ---- *)
(* ============================================================ *)
(* PLC_PRG — главная программа (MainTask)                       *)
(* ============================================================ *)
(* === ДДЮТ:ИЗМЕНЕНО — порядок вызова ===                      *)
(* PR200 и резерв полива СПК на ДДЮТ ОТКЛЮЧЕНЫ (закомментированы)*)
(* Вернуть PR200: раскомментировать PRG_PR200() + поднять канал  *)
(* slave в дереве Modbus. Файлы PRG_PR200/PRG_PolivSPK НЕ удалены.*)
(* ============================================================ *)
PROGRAM PLC_PRG
VAR
END_VAR
PRG_IO();         (* распаковка DI, сборка маски DO *)
PRG_Fountain();   (* автоматика фонтана, дозация, заслонка *)

(* === ДДЮТ:УДАЛИТЬ-условно — PR200 пока нет (может появиться) === *)
(* PRG_PR200(); *)

(* === ДДЮТ:УДАЛИТЬ — резерв полива СПК (нет ямы слива) === *)
(* PRG_PolivSPK(); *)

PRG_Pumps();      (* обработка ПЧ-насосов фонтана (COM2) *)
PRG_Errors();     (* подсчёт общих аварий *)

(* ---- PRG_AlarmLogSD.st ---- *)
(* ============================================================ *)
(* PRG_AlarmLogSD — ЖУРНАЛЫ НА SD-КАРТУ (3 файла В МЕСЯЦ) — ДДЮТ *)
(* ============================================================ *)
(* Пишет на SD три отдельных журнала (чтобы записи не путались): *)
(*   • АВАРИИ      → sAlarmLogPath   (alarms-MM-YYYY.log)       *)
(*   • ИЗМЕНЕНИЯ ПЧ → sPumpLogPath    (pump_changes-MM-YYYY.log) *)
(*   • УСТАВКИ     → sSetpointLogPath (setpoints-MM-YYYY.log)   *)
(*                                                              *)
(* === НОВОЕ: ПОМЕСЯЧНЫЕ ФАЙЛЫ ==============================    *)
(* Имя файла содержит месяц и год, поэтому 1-го числа нового     *)
(* месяца путь меняется САМ, и старый автомат (OPEN → если нет   *)
(* файла, то CREATE + BOM) создаёт новый файл без единой строчки *)
(* дополнительной логики. Отдельного «переключателя месяца» нет  *)
(* специально: любая пропущенная граница (ПЛК был выключен,      *)
(* карту вынимали) отрабатывается сама собой при первой записи.  *)
(*                                                              *)
(* === НОВОЕ: КОНТРОЛЬ МЕСТА ================================    *)
(* FB_SdSpaceGuard раз в tSdCheckPeriod (по умолчанию час), при  *)
(* смене месяца и после серии неудачных записей удаляет три файла *)
(* самого старого месяца, если журналы переросли квоту:            *)
(*     квота = ёмкость карты − 100 МБ резерва − чужие файлы        *)
(* Файл текущего месяца удалить нельзя ни при каких условиях.      *)
(*                                                               *)
(* ЁМКОСТЬ КАРТЫ ОПРЕДЕЛЯЕТСЯ АВТОМАТИЧЕСКИ — FB_SdCardSize        *)
(* читает размер раздела у ядра (/sys/block/...). Номинал из       *)
(* выпадающего списка на экране (iSdCardSize) — только запасной    *)
(* вариант, если автоопределение не сработало. Кнопок нет.         *)
(*                                                              *)
(* Строка: "чч:мм дд.мм.гггг - текст" (аварии) либо готовая      *)
(* строка журнала (ПЧ/уставки). WSTRING/UTF-16LE + BOM.         *)
(*                                                              *)
(* Аварии детектируются здесь СТРОГО ПО ФРОНТУ FALSE→TRUE: пока  *)
(* авария висит, повторных записей нет. Изменения ПЧ/уставок     *)
(* кладут строку в GVL_Fountain.awsSdPumpQ / awsSdSetpQ прямо из *)
(* F_PumpLogWrite / F_FountainLogWrite — здесь только пишем.     *)
(*                                                              *)
(* Один автомат обслуживает 3 файла (приоритет: аварии → ПЧ →    *)
(* уставки). ФБ CAA File асинхронные. Тип дескриптора            *)
(* FILE.CAA.HANDLE. SD FAT16/FAT32 MBR, /mnt/ufs/media/mmcblk0p1.*)
(* Пока сторож места занят (fbGuard.xBusy) — новая строка не     *)
(* начинается, строки ждут в очередях.                           *)
(* ============================================================ *)
PROGRAM PRG_AlarmLogSD
VAR CONSTANT
    cAlarmCnt       : INT := 12;   // сколько аварий отслеживаем (ДДЮТ)
    cQSize          : INT := 20;
    cWriteFailForce : INT := 3;    // столько неудачных записей подряд =
                                   // карта полна → удалить старый месяц
END_VAR
VAR
    (* --- Аварии: состояние + названия --- *)
    axAlarmNow  : ARRAY[1..cAlarmCnt] OF BOOL;
    axAlarmPrev : ARRAY[1..cAlarmCnt] OF BOOL;
    awsAlarmName : ARRAY[1..cAlarmCnt] OF WSTRING(60) := [
        "Сухой ход",
        "Сухой ход реле",
        "Добор — исчерпаны попытки",
        "Альгицид (защ.таймер)",
        "Биопаг (защ.таймер)",
        "pH реле",
        "Альгицид реле",
        "Биопаг реле",
        "Связь ПЧ1",
        "Связь ПЧ2",
        "Связь МВ-Д",
        "Связь МУ"];

    (* --- Локальная очередь аварий (сырые строки) --- *)
    awsAlarmQ : ARRAY[1..cQSize] OF WSTRING(120);
    iAQHead : INT;  iAQTail : INT;  iAQCount : INT;

    (* --- Конечный автомат --- *)
    iState     : INT;
    wsLineOut  : WSTRING(122);
    sActivePath : STRING(80);
    wBom       : WORD := 16#FEFF;

    fbFileOpen  : FILE.Open;
    fbFileWrite : FILE.Write;
    fbFileFlush : FILE.Flush;
    fbFileClose : FILE.Close;
    hFile       : FILE.CAA.HANDLE;

    iWrittenCnt : INT;
    iDroppedCnt : INT;

    i          : INT;
    wsTimeStamp : WSTRING(24);
    wsHH : WSTRING(4);  wsMM : WSTRING(4);
    wsDD : WSTRING(4);  wsMo : WSTRING(4);  wsYY : WSTRING(6);

    (* --- Помесячные файлы --- *)
    iLogYear      : INT;    // год/месяц, в которые сейчас пишем
    iLogMonth     : INT;
    iLogYearPrev  : INT;    // 0 при старте → пути соберутся в 1-м же цикле
    iLogMonthPrev : INT;

    (* --- Сторож места на карте --- *)
    fbGuard         : FB_SdSpaceGuard;
    fbCardSize      : FB_SdCardSize;   // автоопределение ёмкости карты
    tonSdCheck      : TON;
    xGuardTrig      : BOOL;
    xGuardStart     : BOOL;
    xCapTrig        : BOOL;   // перечитать ёмкость карты
    xGuardForceAuto : BOOL;   // авто-форс: карта полна (серия отказов записи)
    iWriteFailCnt   : INT;    // неудачных записей подряд
END_VAR

(* ============================================================ *)
(* 1. КАРТА АВАРИЙ (порядок = порядок названий)                 *)
(* ============================================================ *)
axAlarmNow[1]  := xDryRunAlarm;
axAlarmNow[2]  := xDryRunRelayAlarm;
axAlarmNow[3]  := xRefillAttemptsAlarm;
axAlarmNow[4]  := xAlgAlarm;
axAlarmNow[5]  := xBioAlarm;
axAlarmNow[6]  := xPhRelayAlarm;
axAlarmNow[7]  := xAlgRelayAlarm;
axAlarmNow[8]  := xBioRelayAlarm;
axAlarmNow[9]  := xPumpCommError[1];
axAlarmNow[10] := xPumpCommError[2];
axAlarmNow[11] := xMV110_Error;
axAlarmNow[12] := xMU110_Error;

(* ============================================================ *)
(* 2. МЕТКА ВРЕМЕНИ "чч:мм дд.мм.гггг"                          *)
(* ============================================================ *)
wsHH := INT_TO_WSTRING(iCurrentHour);   IF iCurrentHour   < 10 THEN wsHH := WCONCAT("0", wsHH); END_IF;
wsMM := INT_TO_WSTRING(iCurrentMinute); IF iCurrentMinute < 10 THEN wsMM := WCONCAT("0", wsMM); END_IF;
wsDD := INT_TO_WSTRING(iCurrentDay);    IF iCurrentDay    < 10 THEN wsDD := WCONCAT("0", wsDD); END_IF;
wsMo := INT_TO_WSTRING(iCurrentMonth);  IF iCurrentMonth  < 10 THEN wsMo := WCONCAT("0", wsMo); END_IF;
wsYY := INT_TO_WSTRING(iCurrentYear);
wsTimeStamp := WCONCAT(wsHH, WCONCAT(":", WCONCAT(wsMM, WCONCAT(" ",
               WCONCAT(wsDD, WCONCAT(".", WCONCAT(wsMo, WCONCAT(".", wsYY))))))));

(* ============================================================ *)
(* 3. ФРОНТ АВАРИИ → строка в локальную очередь аварий          *)
(* ============================================================ *)
FOR i := 1 TO cAlarmCnt DO
    IF axAlarmNow[i] AND NOT axAlarmPrev[i] THEN
        IF xAlarmLogSDEnable THEN
            IF iAQCount < cQSize THEN
                iAQTail := (iAQTail MOD cQSize) + 1;
                awsAlarmQ[iAQTail] := WCONCAT(wsTimeStamp, WCONCAT(" - ", awsAlarmName[i]));
                iAQCount := iAQCount + 1;
            ELSE
                iDroppedCnt := iDroppedCnt + 1;
            END_IF;
        END_IF;
    END_IF;
    axAlarmPrev[i] := axAlarmNow[i];
END_FOR;

(* ============================================================ *)
(* 4. ПУТИ ФАЙЛОВ ТЕКУЩЕГО МЕСЯЦА                               *)
(* ============================================================ *)
(* Если RTC ещё не готов или сбит (села батарейка) — год выйдет  *)
(* за 2000..2199. Писать в "alarms-01-1970.log" нельзя (такой     *)
(* месяц не разберётся обратно и файл станет неудаляемым), поэтому*)
(* весь «бесчасовой» период сваливаем в один файл 01-2000. Он     *)
(* заведомо самый старый по ключу, то есть удалится первым, когда *)
(* место кончится, — и при этом защищён как «текущий», пока RTC   *)
(* не починят.                                                   *)
IF iCurrentYear >= 2000 AND iCurrentYear <= 2199
   AND iCurrentMonth >= 1 AND iCurrentMonth <= 12 THEN
    iLogYear  := iCurrentYear;
    iLogMonth := iCurrentMonth;
    xSdRtcBad := FALSE;
ELSE
    iLogYear  := 2000;
    iLogMonth := 1;
    xSdRtcBad := TRUE;
END_IF;

IF iLogYear <> iLogYearPrev OR iLogMonth <> iLogMonthPrev THEN
    sAlarmLogPath    := F_SdLogPath(sSdLogDir, sAlarmLogPrefix, iLogYear, iLogMonth);
    sPumpLogPath     := F_SdLogPath(sSdLogDir, sPumpLogPrefix,  iLogYear, iLogMonth);
    sSetpointLogPath := F_SdLogPath(sSdLogDir, sSetpLogPrefix,  iLogYear, iLogMonth);
    iLogYearPrev     := iLogYear;
    iLogMonthPrev    := iLogMonth;
    xGuardTrig       := TRUE;    // новый месяц — сразу проверить место
    xCapTrig         := TRUE;    // и заодно перечитать ёмкость карты
END_IF;

(* ============================================================ *)
(* 5. СТОРОЖ МЕСТА НА КАРТЕ                                     *)
(* ============================================================ *)
(* Периодический тик (самосброс: Q взводится на 1 цикл за период) *)
tonSdCheck(IN := NOT tonSdCheck.Q, PT := tSdCheckPeriod);
IF tonSdCheck.Q THEN
    xCapTrig   := TRUE;
    xGuardTrig := TRUE;
END_IF;

(* --- ЁМКОСТЬ КАРТЫ ---                                           *)
(* Сначала пробуем определить её САМИ (FB_SdCardSize читает размер *)
(* раздела у ядра). Получилось — номинал из списка не нужен вообще. *)
(* Не получилось — берём выбранный на экране номинал.               *)
fbCardSize(xTrigger := xCapTrig AND (iState = 0) AND NOT fbGuard.xBusy,
           sSysPath := sSdCardSysPath);
IF fbCardSize.xBusy THEN
    xCapTrig := FALSE;
END_IF;

xSdCapAuto       := fbCardSize.xValid;
udiSdCapAutoMB   := fbCardSize.udiCapacityMB;
udiSdCardSectors := fbCardSize.udiSectors;

IF iSdCardSize < 0 THEN iSdCardSize := 0; END_IF;
IF iSdCardSize > 6 THEN iSdCardSize := 6; END_IF;

IF xSdCapAuto THEN
    udiSdUsableMB := udiSdCapAutoMB;
ELSE
    udiSdUsableMB := audiSdCardMB[iSdCardSize];
END_IF;

(* АВАРИЙНЫЙ ФОРС. Если запись не проходит подряд cWriteFailForce  *)
(* раз — карта реально полна, что бы ни говорил расчёт по номиналу *)
(* (например, в списке выбрали 32 ГБ, а стоит карта на 16). Тогда  *)
(* удаляем самый старый месяц безусловно. Одиночный сбой записи к  *)
(* удалению НЕ приводит — только серия подряд.                     *)
IF iWriteFailCnt >= cWriteFailForce THEN
    xGuardTrig      := TRUE;
    xGuardForceAuto := TRUE;
    iWriteFailCnt   := 0;
END_IF;

(* Запускаем сторожа ТОЛЬКО когда автомат записи стоит в IDLE:     *)
(* так исключено удаление файла при открытом дескрипторе.          *)
xGuardStart := xGuardTrig AND xAlarmLogSDEnable
               AND (iState = 0) AND NOT fbGuard.xBusy AND NOT fbCardSize.xBusy;

fbGuard(xTrigger      := xGuardStart,
        xForce        := xGuardForceAuto,
        sDir          := sSdLogDir,
        sPrefix1      := sAlarmLogPrefix,
        sPrefix2      := sPumpLogPrefix,
        sPrefix3      := sSetpLogPrefix,
        udiUsableMB   := udiSdUsableMB,
        udiFreeMinMB  := udiSdFreeMinMB,
        iCurYear      := iLogYear,
        iCurMonth     := iLogMonth);

IF fbGuard.xBusy THEN
    xGuardTrig      := FALSE;
    xGuardForceAuto := FALSE;
END_IF;

(* Диагностика на экран *)
udiSdQuotaMB       := fbGuard.udiQuotaMB;
udiSdOursMB        := fbGuard.udiOursMB;
udiSdUsedMB        := fbGuard.udiUsedMB;
udiSdForeignMB     := fbGuard.udiForeignMB;
udiSdOldestMB      := fbGuard.udiOldestMB;
xSdNothingToDelete := fbGuard.xNothingToDelete;
xSdLogQuotaStop    := fbGuard.xQuotaStop;
xSdCleanupFault    := fbGuard.xFault;
iSdDeletedTotal    := fbGuard.iDeletedTotal;
sSdLastDeleted     := fbGuard.sLastDeleted;

(* ============================================================ *)
(* 6. КОНЕЧНЫЙ АВТОМАТ: пишет по очереди 3 файла                *)
(*    приоритет: аварии → изменения ПЧ → уставки               *)
(* ============================================================ *)
(* Запись стоит, пока сторож занят (иначе он удалял бы файл с    *)
(* открытым дескриптором) ИЛИ пока поднят xQuotaStop — последний *)
(* рубеж защиты карты: наши журналы упёрлись в квоту, а удалять   *)
(* уже нечего. Строки при этом копятся в очередях, лишние         *)
(* считаются в iDroppedCnt; журналы на экране ведутся как обычно. *)
IF NOT fbGuard.xBusy AND NOT fbCardSize.xBusy AND NOT fbGuard.xQuotaStop THEN

CASE iState OF

    0:  (* IDLE — выбрать непустую очередь, взять строку, начать *)
        IF xAlarmLogSDEnable THEN
            IF iAQCount > 0 THEN
                iAQHead := (iAQHead MOD cQSize) + 1;
                wsLineOut := WCONCAT(awsAlarmQ[iAQHead], "$R$N");
                iAQCount := iAQCount - 1;
                sActivePath := sAlarmLogPath;
                iState := 1;
            ELSIF iSdPumpQCount > 0 THEN
                iSdPumpQHead := (iSdPumpQHead MOD 20) + 1;
                wsLineOut := WCONCAT(awsSdPumpQ[iSdPumpQHead], "$R$N");
                iSdPumpQCount := iSdPumpQCount - 1;
                sActivePath := sPumpLogPath;
                iState := 1;
            ELSIF iSdSetpQCount > 0 THEN
                iSdSetpQHead := (iSdSetpQHead MOD 20) + 1;
                wsLineOut := WCONCAT(awsSdSetpQ[iSdSetpQHead], "$R$N");
                iSdSetpQCount := iSdSetpQCount - 1;
                sActivePath := sSetpointLogPath;
                iState := 1;
            END_IF;
        END_IF;

    1:  (* OPEN на дозапись *)
        fbFileOpen(xExecute := TRUE, sFileName := sActivePath, eFileMode := FILE.MODE.MAPPD);
        IF fbFileOpen.xDone THEN
            hFile := fbFileOpen.hFile;
            fbFileOpen(xExecute := FALSE);
            iState := 3;
        ELSIF fbFileOpen.xError THEN
            IF fbFileOpen.eError = FILE.ERROR.NOT_EXIST THEN
                fbFileOpen(xExecute := FALSE);
                iState := 2;
            ELSE
                fbFileOpen(xExecute := FALSE);
                iState := 9;
            END_IF;
        END_IF;

    2:  (* CREATE — MWRITE создаёт файл *)
        fbFileOpen(xExecute := TRUE, sFileName := sActivePath, eFileMode := FILE.MODE.MWRITE);
        IF fbFileOpen.xDone THEN
            hFile := fbFileOpen.hFile;
            fbFileOpen(xExecute := FALSE);
            iState := 6;
        ELSIF fbFileOpen.xError THEN
            fbFileOpen(xExecute := FALSE);
            iState := 9;
        END_IF;

    6:  (* WRITE_BOM — метка UTF-16LE в начало нового файла *)
        fbFileWrite(xExecute := TRUE, hFile := hFile, pBuffer := ADR(wBom), szSize := UDINT#2);
        IF fbFileWrite.xDone THEN
            fbFileWrite(xExecute := FALSE);
            iState := 3;
        ELSIF fbFileWrite.xError THEN
            fbFileWrite(xExecute := FALSE);
            xSdWriteFault := TRUE;
            xGuardTrig    := TRUE;
            iWriteFailCnt := iWriteFailCnt + 1;      // не пишется — проверить место
            iState := 5;
        END_IF;

    3:  (* WRITE — строка WSTRING, размер = WLEN*2 байт *)
        fbFileWrite(xExecute := TRUE, hFile := hFile,
                    pBuffer := ADR(wsLineOut), szSize := INT_TO_UDINT(WLEN(wsLineOut) * 2));
        IF fbFileWrite.xDone THEN
            fbFileWrite(xExecute := FALSE);
            iWrittenCnt := iWrittenCnt + 1;
            xSdWriteFault := FALSE;
            iWriteFailCnt := 0;         // запись прошла — серия отказов сброшена
            iState := 4;
        ELSIF fbFileWrite.xError THEN
            fbFileWrite(xExecute := FALSE);
            xSdWriteFault := TRUE;
            xGuardTrig    := TRUE;
            iWriteFailCnt := iWriteFailCnt + 1;
            iState := 5;
        END_IF;

    4:  (* FLUSH *)
        fbFileFlush(xExecute := TRUE, hFile := hFile);
        IF fbFileFlush.xDone OR fbFileFlush.xError THEN
            fbFileFlush(xExecute := FALSE);
            iState := 5;
        END_IF;

    5:  (* CLOSE *)
        fbFileClose(xExecute := TRUE, hFile := hFile);
        IF fbFileClose.xDone OR fbFileClose.xError THEN
            fbFileClose(xExecute := FALSE);
            iState := 0;
        END_IF;

    9:  (* DROP — ошибка открытия/создания, едем дальше *)
        xSdWriteFault := TRUE;
        xGuardTrig    := TRUE;
        iWriteFailCnt := iWriteFailCnt + 1;
        iState := 0;

END_CASE;

END_IF;

(* ---- PRG_Errors.st ---- *)
(* ============================================================ *)
(* PRG_Errors — ЕДИНЫЙ подсчёт аварий + статус системы          *)
(* Проект ДДЮТ (на основе Fontan_V1 / Саки Пруд).                *)
(*                                                                *)
(* === ДДЮТ:ИЗМЕНЕНО === Убраны аварии несуществующего            *)
(* оборудования (перелив/датчик/протечка/концевики/свет/резерв   *)
(* полива/МВ-8А). Добавлены: биопаг (в Саки не считался — это     *)
(* был пробел, тут исправлено) и три аварии реле обратной связи   *)
(* дозаторов (pH/альгицид/биопаг).                                *)
(* ============================================================ *)
PROGRAM PRG_Errors
VAR
    i : INT;
END_VAR

iErrors         := 0;
iErrorsPumps    := 0;
iErrorsModules  := 0;
iErrorsFountain := 0;
iWorkCount      := 0;
iStopCount      := 0;

(* ============================================================ *)
(* 1. АВАРИИ НАСОСОВ ПЧ (счётчик iErrorsPumps)                 *)
(* ============================================================ *)
FOR i := 1 TO cPumpCount DO
    IF xPumpAlarm[i] AND NOT xPumpCommError[i] THEN
        iErrorsPumps := iErrorsPumps + 1;
    END_IF;
    IF xPumpWork[i] THEN iWorkCount := iWorkCount + 1; END_IF;
    IF xPumpStop[i] THEN iStopCount := iStopCount + 1; END_IF;
END_FOR;

(* ============================================================ *)
(* 2. АВАРИИ СВЯЗИ МОДУЛЕЙ (счётчик iErrorsModules)             *)
(* ============================================================ *)
FOR i := 1 TO cPumpCount DO
    IF xPumpCommError[i] THEN
        iErrorsModules := iErrorsModules + 1;
    END_IF;
END_FOR;
IF xMV110_Error THEN iErrorsModules := iErrorsModules + 1; END_IF;  // МВ110-16Д
IF xMU110_Error THEN iErrorsModules := iErrorsModules + 1; END_IF;  // МУ110-16Р
(* === ДДЮТ:УДАЛИТЬ === нет модуля МВ110-8А (аналоговый) *)
(* IF xMV110_8A_Error THEN iErrorsModules := iErrorsModules + 1; END_IF; *)

(* ============================================================ *)
(* 3. АВАРИИ АВТОМАТИКИ ФОНТАНА (iErrorsFountain)               *)
(* ============================================================ *)
IF xDryRunAlarm         THEN iErrorsFountain := iErrorsFountain + 1; END_IF;  // сухой ход (вычисляемый)
IF xDryRunRelayAlarm    THEN iErrorsFountain := iErrorsFountain + 1; END_IF;  // ДДЮТ: DO13/DI6 расхождение
IF xRefillAttemptsAlarm THEN iErrorsFountain := iErrorsFountain + 1; END_IF;  // ДДЮТ: исчерпаны попытки добора
IF xAlgAlarm            THEN iErrorsFountain := iErrorsFountain + 1; END_IF;  // альгицид (защ.таймер)
IF xBioAlarm            THEN iErrorsFountain := iErrorsFountain + 1; END_IF;  // биопаг (защ.таймер) — ДДЮТ:добавлено
IF xPhRelayAlarm       THEN iErrorsFountain := iErrorsFountain + 1; END_IF;  // ДДЮТ: реле pH нет подтверждения
IF xAlgRelayAlarm      THEN iErrorsFountain := iErrorsFountain + 1; END_IF;  // ДДЮТ: реле альгицида
IF xBioRelayAlarm      THEN iErrorsFountain := iErrorsFountain + 1; END_IF;  // ДДЮТ: реле биопага

(* === ДДЮТ:УДАЛИТЬ === аварии несуществующего оборудования *)
(*
IF xAlarmOverflow      THEN iErrorsFountain := iErrorsFountain + 1; END_IF;
IF xAlarmWaterSensor   THEN iErrorsFountain := iErrorsFountain + 1; END_IF;
IF xDamperAlarm        THEN iErrorsFountain := iErrorsFountain + 1; END_IF;
IF xDamperSensorFault  THEN iErrorsFountain := iErrorsFountain + 1; END_IF;
IF xLeakAlarm          THEN iErrorsFountain := iErrorsFountain + 1; END_IF;
IF xLightFault         THEN iErrorsFountain := iErrorsFountain + 1; END_IF;
IF xSpkErrPereliv      THEN iErrorsFountain := iErrorsFountain + 1; END_IF;
IF xSpkErrDobor        THEN iErrorsFountain := iErrorsFountain + 1; END_IF;
IF xSpkErrPoliv        THEN iErrorsFountain := iErrorsFountain + 1; END_IF;
*)

(* ============================================================ *)
(* 4. ОБЩИЙ СЧЁТЧИК ВСЕХ АВАРИЙ + ЕДИНЫЙ ФЛАГ                  *)
(* ============================================================ *)
iErrors   := iErrorsPumps + iErrorsModules + iErrorsFountain;
xAnyAlarm := (iErrors > 0);

xSystemState := NOT xAnyAlarm;
IF xSystemState THEN
    sSystemStateText := "Система: ОК";
ELSE
    sSystemStateText := "Авария";
END_IF;
